(* IEC 61131-3 sources: verifaps-lib/geteta/examples/issue2, 1 file *)

(* ---- issue2.st ---- *)
TYPE
  var_enumD : (var_literalOne, var_literalTwo);
END_TYPE

PROGRAM var_constantprogram
  VAR_INPUT
    var_A : INT;
    var_B : BOOL;
  END_VAR

  VAR_OUTPUT
    var_C : INT;
    var_D : var_enumD;
  END_VAR

  var_C := 52;
END_PROGRAM
